FUNCTION_BLOCK CarbonDioxideSensor EXTENDS Device IMPLEMENTS SHLib.IInputDevice
VAR
	_CarbonDioxideLevel : WORD := 800;
END_VAR

{attribute 'monitoring' := 'call'}
PROPERTY CarbonDioxideLevel : WORD
GET
CarbonDioxideLevel := _CarbonDioxideLevel;
END_GET
END_PROPERTY

{attribute 'monitoring' := 'call'}
PROPERTY Name : STRING
GET
Name := 'OxygenSensor';
END_GET
END_PROPERTY

METHOD ReadInputs
// handle value from terminal here
END_METHOD

END_FUNCTION_BLOCK

(* stored: Version 1.1.0.1
   POU CarbonDioxideSensor: Id {e1272fbc-4237-4208-a038-78ed9d5f74fb}, SpecialFunc None
   Property CarbonDioxideLevel: Id {0c6e80c7-98d8-4516-933b-6944d6c6aab0}
   Get Get: Id {f76bd113-b113-4150-89e5-ce4c15d93ba9}
   Property Name: Id {7626f8d8-020e-4fa5-98fd-9a9237729a65}
   Get Get: Id {628b7714-3354-4018-9b95-9ddd8ae3d138}
   Method ReadInputs: Id {aa64c8a8-f985-46ea-83c3-4a2fce2ee799} *)
